Universal Robots URScript: Robot 3 12_10.script

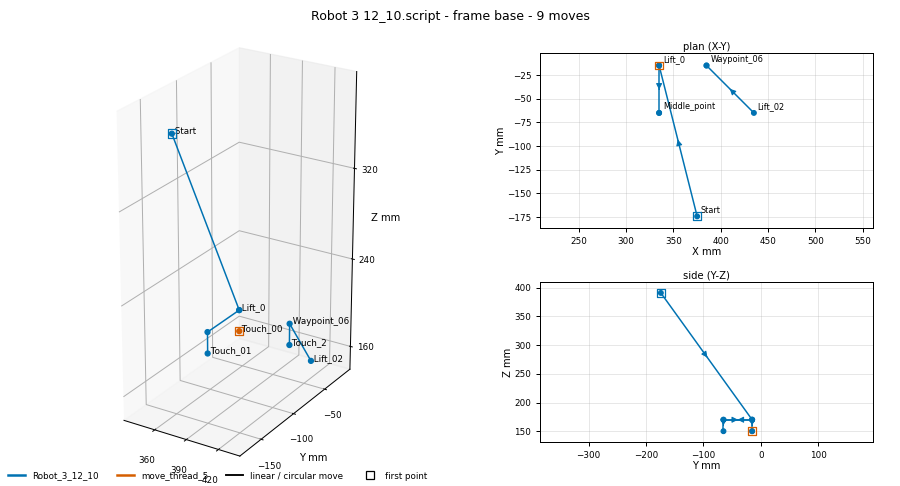
[picture p0: tool path of Robot 3 12_10.script in frame base, 9 of 16 moves have a stored position in this frame; points joined in program order, loops and branches not executed]
def Robot_3_12_10():
  set_tcp(p[0.0,0.0,0.0,0.0,0.0,0.0])
  set_safety_mode_transition_hardness(1)
  step_count_74a58e22_dc11_493a_940f_6be2cdcaf4fc = 0.0
  thread Step_Counter_Thread_ecd05ca1_44cd_422d_8c53_38ca33f79cc8():
    while (True):
      step_count_74a58e22_dc11_493a_940f_6be2cdcaf4fc = step_count_74a58e22_dc11_493a_940f_6be2cdcaf4fc + 1.0
      sync()
    end
  end
  run Step_Counter_Thread_ecd05ca1_44cd_422d_8c53_38ca33f79cc8()
  set_target_payload(0.990000, [-0.002000, -0.006000, 0.057000], [0.001514, 0.001514, 0.001514, 0.000000, 0.000000, 0.000000])
  modbus_add_signal("192.168.12.20", 255, 1001, 2, "MODBUS_1", False)
  modbus_set_signal_update_frequency("MODBUS_1", 10)
  modbus_add_signal("192.168.12.20", 255, 1003, 3, "MODBUS_2", False)
  modbus_set_signal_update_frequency("MODBUS_2", 10)
  modbus_add_signal("192.168.12.20", 255, 1005, 2, "MODBUS_3", False)
  modbus_set_signal_update_frequency("MODBUS_3", 10)
  modbus_add_signal("192.168.12.20", 255, 1008, 2, "MODBUS_4", False)
  modbus_set_signal_update_frequency("MODBUS_4", 10)
  modbus_add_signal("192.168.12.20", 255, 1007, 3, "MODBUS_5", False)
  modbus_set_signal_update_frequency("MODBUS_5", 10)
  modbus_set_runstate_dependent_choice("MODBUS_2",0)
  modbus_set_runstate_dependent_choice("MODBUS_5",0)
  set_gravity([0.0, 0.0, 9.82])
  set_tool_communication(True, 1000000, 2, 1, 1.5, 3.5)
  set_tool_output_mode(0)
  set_tool_digital_output_mode(0, 1)
  set_tool_digital_output_mode(1, 1)
  set_tool_voltage(24)
  set_standard_analog_input_domain(0, 1)
  set_standard_analog_input_domain(1, 1)
  set_tool_analog_input_domain(0, 1)
  set_tool_analog_input_domain(1, 1)
  set_analog_outputdomain(0, 0)
  set_analog_outputdomain(1, 0)
  set_input_actions_to_default()
  global Plane_1=p[0.5,0.0,0.07,-3.667604942726106E-16,3.141592653589793,-5.847522753981501E-16]
  # begin: URCap Installation Node
  #   Source: OnRobot, 5.14.0, OnRobot A/S
  #   Type: OnRobot Setup
  if (False):
  end
  ON_CONN_SHIFT_BOOL = 64
  ON_CONN_SHIFT_INT = 24
  ON_CONN_SHIFT_FLOAT = 24
  ON_CONN_REG_SUM_BOOL = 0
  ON_CONN_REG_SUM_INT = 1
  ON_CONN_REG_SUM_FLOAT = 0
  ON_TOOL_SHIFT_BOOL = 64
  ON_TOOL_SHIFT_INT = 25
  ON_TOOL_SHIFT_FLOAT = 24
  ON_TOOL_SHIFT_BOOL_ARR = [64, 64, 64]
  ON_TOOL_SHIFT_INT_ARR = [25, 25, 25]
  ON_TOOL_SHIFT_FLOAT_ARR = [24, 24, 24]
  ON_TOOL_REG_SUM_BOOL = 0
  ON_TOOL_REG_SUM_INT = 0
  ON_TOOL_REG_SUM_FLOAT = 0
  ON_REGISTERS_SPEEDL_FLOAT = 0
  ON_REG_USE_TOOL = False
  ON_DI_SINGLE = 0
  ON_DI_PRIMARY = 1
  ON_DI_SECONDARY = 2
  ON_DI_DUAL = 3
  on_robot_type = 10
  on_robot_cycle = 2.0
  on_conn_ip = "localhost"
  on_tool_ip = "localhost"
  on_device_socket_port = 51234
  on_conn_xmlrpc = rpc_factory("xmlrpc", "http://localhost:41414")
  on_tool_xmlrpc = rpc_factory("xmlrpc", "http://localhost:41414")
  on_RPC = rpc_factory("xmlrpc", "http://127.0.0.1:31416")
  ON_DEBUG_LOG = False
  on_isMetric = True
  on_toolConnector = True
  on_ioqc = False
  on_dual = False
  on_computebox = False
  on_devices = 0
  on_gripper = [False, False, False]
  on_custom_tcp_id = "none"
  on_custom_tcp_enabled = False
  on_ft = False
  #======    OnRobot Globals    ======#

  ON_MATH_PI=3.141593
  ON_ZEROPOSE=p[0.0,0.0,0.0,0.0,0.0,0.0]
  ON_ZEROFRAME=p[0.0,0.0,0.0,0.0,0.0,0.0]
  ON_ZERO3D=[0.0,0.0,0.0]
  ON_ZERO6D=[0.0,0.0,0.0,0.0,0.0,0.0]
  ON_ZERO8D=[0.0,0.0,0.0,0.0,0.0,0.0,0.0,0.0]
  ON_FALSE3D=[False,False,False]
  ON_FALSE6D=[False,False,False,False,False,False]
  ON_FALSE8D=[False,False,False,False,False,False,False,False]
  global on_return=0
  on_speedL=ON_ZERO6D
  on_speedBase=ON_ZERO6D
  on_speedVect=ON_ZERO6D
  on_speedExtra=ON_ZERO6D
  on_speedCB=ON_ZERO6D
  on_speedGecko=ON_ZERO6D
  on_RTDE_error=0
  on_RTDE_tool_error=0
  on_dataProcess_thrd=0
  ON_DEVICE_ID_MISSING=0
  ON_INIT_WATCHDOG_HZ=5
  ON_INIT_TIMEOUT=500
  on_robot_TCP_offset=ON_ZEROFRAME
  on_tcp_offset_actual=ON_ZEROFRAME
  on_cog_actual=ON_ZEROFRAME
  on_mass_actual=0.0
  on_robot_mount=[0.0,0.0]

  #======    End of OnRobot Globals    ======#
  #======    OnRobot Interface Messages    ======#

  on_devices_primary_log="OnRobot Devices"
  on_devices_secondary_log="OnRobot Secondary Device"
  on_program_halted="<br>Program halted."
  on_device_error_title="OnRobot - Device error"
  on_install_error="OnRobot Setup is not correct.<br>Check the status in the OnRobot Setup page in the Installation Tab.<br>Program halted."
  on_device_missing="No device connected.<br>Program halted."
  cb_device_missing="No OnRobot Compute Box connected.<br>Program halted."
  ft_device_missing="No OnRobot FT sensor or license detected.<br>Program halted."
  hex_device_missing="No HEX sensor connected.<br>Program halted."
  rg2ft_device_missing="No RG2-FT gripper connected.<br>Program halted."
  rg_device_missing="No RG gripper connected.<br>Program halted."
  vg_device_missing="No VG gripper connected.<br>Program halted."
  gg_device_missing="No Gecko Gripper connected.<br>Program halted."
  sg_device_missing="No Soft Gripper connected.<br>Program halted."
  tfg_device_missing="No 3FG gripper connected.<br>Program halted."
  sdr_device_missing="No OnRobot Sander connected.<br>Program halted."
  twofg_device_missing="No 2FG gripper connected.<br>Program halted."
  vgp_device_missing="No VGP gripper connected.<br>Program halted."
  mg_device_missing="No Magnetic Gripper connected.<br>Program halted."
  fgp_device_missing="No 2FGP20 Gripper connected.<br>Program halted."
  on_xmlrpc_start_ip="Connecting to OnRobot XML-RPC Server:"
  on_java_comm_error_textmsg_title="OnRobot - Communication error:"
  on_java_comm_controlsocket_open_error="Socket 'javaSocket' opening was unsuccessful."
  on_java_comm_error_title="OnRobot - Communication error"
  on_java_comm_socket_open_error="Establishing connection with the URCap was timed out.<br>Check the status in the OnRobot Setup page in the Installation Tab.<br>Program halted."
  on_rtde_feed_error_textmsg_title="OnRobot - RTDE error:"
  on_rtde_feed_error="RTDE feed error. OnRobot device count mismatch.<br>Program halted."
  on_rtde_feed_tool_error="Tool RTDE feed error. OnRobot device count mismatch.<br>Program halted."
  on_rtde_feed_open_error_textmsg="Socket 'rtdeFeed' opening was unsuccessful."
  on_rtde_feed_error_title="OnRobot - RTDE error"
  on_rtde_feed_count_error="Invalid RTDE offset setup detected. Please check RTDE Offsets at the OnRobot Setup page in the Installation Tab.<br>Program halted."
  on_rtde_feed_open_error="Establishing connection with the devices was timed out.<br>Ensure that the OnRobot devices are operational, and check the status in the OnRobot Setup page in the Installation Tab."

  #======    End of OnRobot Interface Messages    ======#
  #======    OnRobot Interface    ======#

  on_portopened_javaSocket=False
  on_rtde_feed_opened=False
  on_dataProcess_running=False
  def on_missing():
  popup(on_device_missing,title=on_device_error_title,error=True,blocking=False)
  halt
  end
  def cb_missing():
  popup(cb_device_missing,title=on_device_error_title,error=True,blocking=False)
  halt
  end
  def ft_missing():
  popup(ft_device_missing,title=on_device_error_title,error=True,blocking=False)
  halt
  end
  def hex_missing():
  popup(hex_device_missing,title=on_device_error_title,error=True,blocking=False)
  halt
  end
  def rg2ft_missing():
  popup(rg2ft_device_missing,title=on_device_error_title,error=True,blocking=False)
  halt
  end
  def rg_missing():
  popup(rg_device_missing,title=on_device_error_title,error=True,blocking=False)
  halt
  end
  def vg_missing():
  popup(vg_device_missing,title=on_device_error_title,error=True,blocking=False)
  halt
  end
  def gg_missing():
  popup(gg_device_missing,title=on_device_error_title,error=True,blocking=False)
  halt
  end
  def sg_missing():
  popup(sg_device_missing,title=on_device_error_title,error=True,blocking=False)
  halt
  end
  def tfg_missing():
  popup(tfg_device_missing,title=on_device_error_title,error=True,blocking=False)
  halt
  end
  def sdr_missing():
  popup(sdr_device_missing,title=on_device_error_title,error=True,blocking=False)
  halt
  end
  def twofg_missing():
  popup(twofg_device_missing,title=on_device_error_title,error=True,blocking=False)
  halt
  end
  def vgp_missing():
  popup(vgp_device_missing,title=on_device_error_title,error=True,blocking=False)
  halt
  end
  def mg_missing():
  popup(mg_device_missing,title=on_device_error_title,error=True,blocking=False)
  halt
  end
  def fgp_missing():
  popup(fgp_device_missing,title=on_device_error_title,error=True,blocking=False)
  halt
  end
  def on_portclose_javaSocket():
  socket_close("javaSocket")
  on_portopened_javaSocket=False
  end
  def on_portopen_javaSocket():
  on_portclose_javaSocket()
  on_portopened_javaSocket=socket_open("127.0.0.1",44005,"javaSocket")
  if not on_portopened_javaSocket:
  textmsg(on_java_comm_error_textmsg_title,on_java_comm_controlsocket_open_error)
  popup(on_java_comm_socket_open_error,title=on_java_comm_error_title,error=True,blocking=False)
  halt
  end
  end
  on_conn_rtde_feed_name="rtdeFeedConn"
  on_tool_rtde_feed_name="rtdeFeedTool"
  def on_rtde_feed_close(rtdeFeedName):
  socket_close(rtdeFeedName)
  on_rtde_feed_opened=False
  end
  def on_rtde_feed_open(deviceIP,rtdeFeedName,regStart,regSum,regSpeedl):
  on_rtde_feed_close(rtdeFeedName)
  if((regStart[0]+regSum[0])>128)or((regStart[1]+regSum[1])>48)or((regStart[2]+regSum[2])>48):
  popup(on_rtde_feed_count_error,title=on_rtde_feed_error_title,error=True,blocking=False)
  textmsg(str_cat("RegStart: ",regStart),str_cat("  -  RegSum: ",regSum))
  halt
  end
  on_rtde_feed_opened=socket_open(deviceIP,on_device_socket_port,rtdeFeedName)
  if not on_rtde_feed_opened:
  on_rtde_feed_opened=socket_open(deviceIP,on_device_socket_port,rtdeFeedName)
  end
  if not on_rtde_feed_opened:
  textmsg(on_rtde_feed_error_textmsg_title,on_rtde_feed_open_error_textmsg)
  popup(on_rtde_feed_open_error,title=on_rtde_feed_error_title,error=True,blocking=False)
  halt
  end
  socket_send_int(regStart[0],rtdeFeedName)
  socket_send_int(regSum[0],rtdeFeedName)
  socket_send_int(regStart[1],rtdeFeedName)
  socket_send_int(regSum[1],rtdeFeedName)
  socket_send_int(regStart[2],rtdeFeedName)
  socket_send_int(regSum[2],rtdeFeedName)
  socket_send_int(regSpeedl,rtdeFeedName)
  socket_send_int(on_devices,rtdeFeedName)
  end
  def on_dataRead():
  enter_critical
  on_RTDE_error=read_input_integer_register(ON_CONN_SHIFT_INT)
  if(ON_REG_USE_TOOL):
  on_RTDE_tool_error=read_input_integer_register(ON_TOOL_SHIFT_INT_ARR[0])
  end
  exit_critical
  end
  def on_set_rtde_watchdog(updateHz=ON_INIT_WATCHDOG_HZ):
  local effect="stop"
  if(updateHz<1):
  effect="ignore"
  end
  watchdog_conn_reg_str=str_cat("input_int_register_",ON_CONN_SHIFT_INT)
  rtde_set_watchdog(watchdog_conn_reg_str,updateHz,effect)
  if(ON_REG_USE_TOOL):
  watchdog_tool_reg_str=str_cat("input_int_register_",ON_TOOL_SHIFT_INT_ARR[0])
  rtde_set_watchdog(watchdog_tool_reg_str,updateHz,effect)
  end
  if ON_DEBUG_LOG:
  local update_str=str_cat(" "+effect+" watchdog set to [Hz]: ",updateHz)
  textmsg(watchdog_conn_reg_str,update_str)
  if(ON_REG_USE_TOOL):
  local update_str=str_cat(" "+effect+" watchdog set to [Hz]: ",updateHz)
  textmsg(watchdog_tool_reg_str,update_str)
  end
  end
  end
  def on_speedCB_get():
  return[on_speedCB[0],on_speedCB[1],on_speedCB[2],on_speedCB[3],on_speedCB[4],on_speedCB[5]]
  end
  def on_speedGecko_get():
  local speedExtra=ON_ZERO6D
  if on_speedl_for_gecko:
  speedExtra=[on_speedGecko[0],on_speedGecko[1],on_speedGecko[2],on_speedGecko[3],on_speedGecko[4],on_speedGecko[5]]
  end
  return speedExtra
  end
  def on_speedGecko_set(speedGecko):
  on_speedGecko=[speedGecko[0],speedGecko[1],speedGecko[2],speedGecko[3],speedGecko[4],speedGecko[5]]
  end
  thread on_dataProcess_thread():
  if ON_DEBUG_LOG:
  textmsg("Starting on_dataRead thread")
  end
  local error=False
  on_dataProcess_running=True
  sync()
  while on_dataProcess_running:
  sync()
  on_dataRead()
  error=on_error((on_RTDE_error<0),on_rtde_feed_error,on_rtde_feed_error_title,error)
  error=on_error((ON_REG_USE_TOOL and(on_RTDE_tool_error<0)),on_rtde_feed_tool_error,on_rtde_feed_error_title,error)
  on_dataProcess_running=not error
  end
  if error:
  halt
  end
  if ON_DEBUG_LOG:
  textmsg("Stopping on_dataRead thread")
  end
  end
  thread on_set_watchdog_thread():
  sleep(2)
  on_set_rtde_watchdog(updateHz=ON_INIT_WATCHDOG_HZ)
  sleep(1/ON_INIT_WATCHDOG_HZ)
  on_dataProcess_running=False
  kill on_dataProcess_thrd
  end

  #======    End of OnRobot Interface    ======#
  #======    OnRobot QC Setup Tool Connector    ======#

  def tc_setup_tool():
  if ON_DEBUG_LOG:
  textmsg("QC Setup Tool Connector start...")
  end
  set_tool_voltage(24)

  set_tool_communication(True,1000000,2,1,1.5,3.5)

  if ON_DEBUG_LOG:
  textmsg("QC Setup Tool Connector end.")
  end
  end

  #======    End of OnRobot QC Setup Tool Connector    ======#
  #======    OnRobot TCP Messages    ======#

  on_tcp_log_msg_default="OnRobot: Robot TCP Offset set to:"
  on_tcp_log_msg_primary="OnRobot: Robot TCP Offset set to Primary:"
  on_tcp_log_msg_secondary="OnRobot: Robot TCP Offset set to Secondary:"

  #======    End of OnRobot TCP Messages    ======#
  #======    OnRobot TCP    ======#

  on_tcp_offset_actual=ON_ZEROFRAME
  on_tcp_offset_primary=ON_ZEROFRAME
  on_tcp_static_primary=ON_ZEROFRAME
  on_tcp_dynamic_primary=ON_ZEROFRAME
  on_tcp_adapters=ON_ZEROFRAME
  on_tcp_qc_primary=ON_ZEROFRAME
  on_tcp_base_primary=ON_ZEROFRAME
  on_tcp_gripper_static_primary=ON_ZEROFRAME
  on_tcp_workpiece_primary=ON_ZEROFRAME
  on_tcp_gripper_dynamic_primary=ON_ZEROFRAME
  on_tcp_gripper_primary=ON_ZEROFRAME
  on_tcp_offset_secondary=ON_ZEROFRAME
  on_tcp_static_secondary=ON_ZEROFRAME
  on_tcp_dynamic_secondary=ON_ZEROFRAME
  on_tcp_qc_secondary=ON_ZEROFRAME
  on_tcp_base_secondary=ON_ZEROFRAME
  on_tcp_gripper_static_secondary=ON_ZEROFRAME
  on_tcp_workpiece_secondary=ON_ZEROFRAME
  on_tcp_gripper_dynamic_secondary=ON_ZEROFRAME
  on_tcp_gripper_secondary=ON_ZEROFRAME
  on_tcp_custom_preset_assigned=False
  on_tcp_custom_preset=ON_ZEROFRAME
  def on_tcp_init_adapters():
  if ON_DEBUG_LOG:
  textmsg("TCP Init Adapters start..")
  end
  enter_critical
  on_tcp_adapters=ON_ZEROFRAME
  local adapterCount=length(on_tcp_adapters_array)
  local i=0
  while(i<adapterCount):
  on_tcp_adapters=pose_trans(on_tcp_adapters,on_tcp_adapters_array[i])
  i=i+1
  end
  exit_critical
  if ON_DEBUG_LOG:
  textmsg("TCP Init Adapters end.")
  end
  end
  def on_tcp_update_primary():
  if ON_DEBUG_LOG:
  textmsg("TCP Update Primary start..")
  end
  on_tcp_gripper_dynamic_primary=p[0.0, 0.0, 0.0, 0.0, 0.0, 0.0]
  enter_critical
  on_tcp_dynamic_primary=pose_trans(on_tcp_static_primary,on_tcp_gripper_dynamic_primary)
  on_tcp_offset_primary=pose_trans(on_tcp_dynamic_primary,on_tcp_workpiece_primary)
  exit_critical
  if ON_DEBUG_LOG:
  textmsg("TCP Update Primary end.")
  end
  end
  def on_tcp_init_primary():
  if ON_DEBUG_LOG:
  textmsg("TCP Init Primary start..")
  end
  enter_critical
  on_tcp_base_primary=pose_trans(on_tcp_adapters,on_tcp_qc_primary)
  on_tcp_static_primary=pose_trans(on_tcp_base_primary,on_tcp_gripper_static_primary)
  exit_critical
  on_tcp_update_primary()
  if ON_DEBUG_LOG:
  textmsg("TCP Init Primary end.")
  end
  end
  def on_tcp_offset_set(TCP_offset):
  if ON_DEBUG_LOG:
  textmsg("TCP Offset set started!")
  end
  on_tcp_offset_send(TCP_offset)
  if(on_follow_tcp):
  set_tcp(TCP_offset)
  end
  on_robot_TCP_offset=TCP_offset
  if ON_DEBUG_LOG:
  textmsg("TCP Offset set to: ",on_robot_TCP_offset)
  end
  end
  def on_tcp_offset_forced_set_actual(isPrimary=True):
  if(not on_follow_tcp):

  local tcp_log_msg=on_tcp_log_msg_default

  textmsg(tcp_log_msg,on_tcp_offset_actual)
  set_tcp(on_tcp_offset_actual)
  end
  end
  def on_tcp_update(isPrimary=True):
  on_tcp_update_primary()

  on_tcp_set_actual_to(isPrimary)
  end
  def on_tcp_set_actual_to(isPrimary=True):

  on_tcp_offset_actual=on_tcp_offset_primary
  if(on_follow_tcp):
  textmsg(on_tcp_log_msg_default,on_tcp_offset_actual)
  end

  on_tcp_active_is_primary=isPrimary
  on_tcp_offset_set(on_tcp_offset_actual)
  end
  def on_tcp_update_workpiece_primary(workpiece_offset):
  if ON_DEBUG_LOG:
  textmsg("TCP Update Tool Primary start..")
  end
  on_tcp_workpiece_primary=workpiece_offset
  on_tcp_update_primary()
  if ON_DEBUG_LOG:
  textmsg("TCP Update Tool Primary end.")
  end
  end
  def on_tcp_workpiece_rpy_get(xyz=[0.0,0.0,0.0],rpy=[0.0,0.0,0.0]):
  local rotvec=rpy2rotvec(rpy)
  local workpiece_offset=p[xyz[0],xyz[1],xyz[2],rotvec[0],rotvec[1],rotvec[2]]
  return workpiece_offset
  end

  def on_tcp_update_workpiece(workpiece_offset,tool_index=0):
  if ON_DEBUG_LOG:
  textmsg("TCP Update Tool start..")
  end
  if(tool_index!=ON_DI_SECONDARY):
  on_tcp_update_workpiece_primary(workpiece_offset)
  local isPrimary=True

  end
  on_tcp_set_actual_to(isPrimary)
  if ON_DEBUG_LOG:
  textmsg("TCP Update Tool end.")
  end
  end
  def on_get_tcp_for(tool_index):
  if tool_index==ON_DI_SECONDARY:
  local actual_tcp=on_tcp_static_secondary
  else:
  local actual_tcp=on_tcp_static_primary
  end
  return actual_tcp
  end
  def on_tcp_custom_unused():
  return ON_ZEROFRAME
  end
  def on_tcp_update_custom():
  if ON_DEBUG_LOG:
  textmsg("TCP Update Custom start..")
  end
  if(on_custom_tcp_enabled):
  on_tcp_custom_unused()
  on_tcp_custom_unused()
  on_tcp_custom_unused()
  on_tcp_custom_unused()

  end
  if ON_DEBUG_LOG:
  textmsg("TCP Update Custom end.")
  end
  end

  #======    End of OnRobot TCP    ======#
  #======    OnRobot Payload Messages    ======#

  on_mass_log_msg="OnRobot: Robot Payload Mass set to:"
  on_cog_log_msg="OnRobot: Robot Payload Center of Gravity set to:"

  #======    End of OnRobot Payload Messages    ======#
  #======    OnRobot Payload    ======#

  on_cog_actual=ON_ZEROFRAME
  on_mass_actual=0.0
  on_cog_primary=ON_ZEROFRAME
  on_cog_L1L2_primary=ON_ZEROFRAME
  on_mass_primary=0.0
  on_mass_L1L2_primary=0.0
  on_cog_adapters=ON_ZEROFRAME
  on_cog_qc_primary=ON_ZEROFRAME
  on_cog_base_primary=ON_ZEROFRAME
  on_cog_gripper_primary=ON_ZEROFRAME
  on_cog_workpiece_primary=ON_ZEROFRAME
  on_mass_adapters=0.0
  on_mass_qc_primary=0.0
  on_mass_base_primary=0.0
  on_mass_gripper_primary=0.0
  on_mass_workpiece_primary=0.0
  on_cog_secondary=ON_ZEROFRAME
  on_mass_secondary=0.0
  on_cog_gripper_secondary=ON_ZEROFRAME
  on_mass_gripper_secondary=0.0
  on_cog_workpiece_secondary=ON_ZEROFRAME
  on_mass_workpiece_secondary=0.0
  ON_LB2KG001=0.45359237/100
  def on_payload_init_adapters():
  if ON_DEBUG_LOG:
  textmsg("TCP Init Adapters start..")
  end
  enter_critical
  on_cog_adapters=ON_ZEROFRAME
  on_mass_adapters=0.0
  local massLAL0Ratio=0
  local adapterAbsCOG=ON_ZEROFRAME
  local tcp_adapter_offset=ON_ZEROFRAME
  local adapterCount=length(on_tcp_adapters_array)
  local i=0
  while(i<adapterCount):
  on_mass_adapters=on_mass_adapters+on_mass_adapters_array[i]
  if(on_mass_adapters<=0):
  massLAL0Ratio=0
  else:
  massLAL0Ratio=on_mass_adapters_array[i]/on_mass_adapters
  end
  adapterAbsCOG=pose_trans(tcp_adapter_offset,on_tcp_adapters_array[i])
  adapterAbsCOG=p[adapterAbsCOG[0],adapterAbsCOG[1],adapterAbsCOG[2],0.0,0.0,0.0]
  on_cog_adapters=interpolate_pose(on_cog_adapters,adapterAbsCOG,massLAL0Ratio)
  on_cog_adapters=p[on_cog_adapters[0],on_cog_adapters[1],on_cog_adapters[2],0.0,0.0,0.0]
  tcp_adapter_offset=pose_trans(tcp_adapter_offset,on_tcp_adapters_array[i])
  i=i+1
  sync()
  end
  exit_critical
  if ON_DEBUG_LOG:
  textmsg("TCP Init Adapters end.")
  end
  end
  def on_payload_update_primary():
  if ON_DEBUG_LOG:
  textmsg("Payload Update Primary start..")
  end
  enter_critical
  on_mass_primary=on_mass_L1L2_primary+on_mass_workpiece_primary
  local massL1L2L3Ratio=on_mass_workpiece_primary/on_mass_primary
  local workpieceAbsCOG=pose_trans(on_tcp_dynamic_primary,on_cog_workpiece_primary)
  workpieceAbsCOG=p[workpieceAbsCOG[0],workpieceAbsCOG[1],workpieceAbsCOG[2],0.0,0.0,0.0]
  on_cog_primary=interpolate_pose(on_cog_L1L2_primary,workpieceAbsCOG,massL1L2L3Ratio)
  on_cog_primary=p[on_cog_primary[0],on_cog_primary[1],on_cog_primary[2],0.0,0.0,0.0]
  exit_critical
  if ON_DEBUG_LOG:
  textmsg("Payload Update Primary end.")
  end
  end
  def on_payload_init_primary():
  if ON_DEBUG_LOG:
  textmsg("Payload Init Primary start..")
  end
  enter_critical
  on_mass_base_primary=on_mass_adapters+on_mass_qc_primary
  local massL0L1Ratio=on_mass_qc_primary/on_mass_base_primary
  on_mass_L1L2_primary=on_mass_base_primary+on_mass_gripper_primary
  local massL1L2Ratio=on_mass_gripper_primary/on_mass_L1L2_primary
  local qcAbsCOG=pose_trans(on_tcp_adapters,on_cog_qc_primary)
  qcAbsCOG=p[qcAbsCOG[0],qcAbsCOG[1],qcAbsCOG[2],0.0,0.0,0.0]
  on_cog_base_primary=interpolate_pose(on_cog_adapters,qcAbsCOG,massL0L1Ratio)
  on_cog_base_primary=p[on_cog_base_primary[0],on_cog_base_primary[1],on_cog_base_primary[2],0.0,0.0,0.0]
  local gripperAbsCOG=pose_trans(on_tcp_base_primary,on_cog_gripper_primary)
  gripperAbsCOG=p[gripperAbsCOG[0],gripperAbsCOG[1],gripperAbsCOG[2],0.0,0.0,0.0]
  on_cog_L1L2_primary=interpolate_pose(on_cog_base_primary,gripperAbsCOG,massL1L2Ratio)
  on_cog_L1L2_primary=p[on_cog_L1L2_primary[0],on_cog_L1L2_primary[1],on_cog_L1L2_primary[2],0.0,0.0,0.0]
  exit_critical
  on_payload_update_primary()
  if ON_DEBUG_LOG:
  textmsg("Payload Init Primary end.")
  end
  end
  def on_payload_update():
  on_payload_update_primary()

  on_mass_actual =on_mass_primary
  on_cog_actual=on_cog_primary

  on_payload_set_actual()
  end
  def on_payload_set_actual():

  on_mass_actual =on_mass_primary
  on_cog_actual=on_cog_primary

  local CoG=[on_cog_actual[0],on_cog_actual[1],on_cog_actual[2]]
  on_payload_set(on_mass_actual,CoG)
  end
  def on_payload_update_workpiece_primary(workpiece_mass=0,workpiece_cog=[0.0,0.0,0.0]):
  if ON_DEBUG_LOG:
  textmsg("Payload Update Workpiece Primary start..")
  end
  on_cog_workpiece_primary=p[workpiece_cog[0],workpiece_cog[1],workpiece_cog[2],0.0,0.0,0.0]
  on_mass_workpiece_primary=workpiece_mass
  on_payload_update_primary()
  if ON_DEBUG_LOG:
  textmsg("Payload Update Workpiece Primary end.")
  end
  end
  def on_payload_set(mass,CoG):
  if ON_DEBUG_LOG:
  textmsg("Payload set started!")
  end
  local center_of_gravity=[CoG[0],CoG[1],CoG[2]]
  on_payload_send(center_of_gravity,mass)
  if(on_isMetric):
  local roundedMass=floor(mass*100+0.5)/100
  else:
  local roundedMass=floor(mass/ON_LB2KG001+0.5)*ON_LB2KG001
  end
  set_payload(roundedMass,center_of_gravity)
  on_mass_actual=roundedMass
  on_cog_actual=p[CoG[0],CoG[1],CoG[2],0.0,0.0,0.0]
  if ON_DEBUG_LOG:
  textmsg("Payload mass, CoG set to: ",str_cat(str_cat(mass,", "),CoG))
  end
  end

  def on_payload_update_secondary():
  end
  def on_payload_init_secondary():
  end

  def on_payload_update_workpiece(workpiece_mass,workpiece_cog=[0.0,0.0,0.0],tool_index=0):
  if ON_DEBUG_LOG:
  textmsg("Payload Update Workpiece start..")
  end
  if(tool_index!=ON_DI_SECONDARY):
  on_cog_workpiece_primary=p[workpiece_cog[0],workpiece_cog[1],workpiece_cog[2],0.0,0.0,0.0]
  on_mass_workpiece_primary=workpiece_mass
  else:
  on_cog_workpiece_secondary=p[workpiece_cog[0],workpiece_cog[1],workpiece_cog[2],0.0,0.0,0.0]
  on_mass_workpiece_secondary=workpiece_mass
  end
  on_payload_update()
  if ON_DEBUG_LOG:
  textmsg("Payload Update Workpiece end.")
  end
  end
  def on_payload_get_cog2tcp_workpiece(tool_index=0):
  if(tool_index!=ON_DI_SECONDARY):
  local cog_tool=[on_tcp_workpiece_primary[0],on_tcp_workpiece_primary[1],on_tcp_workpiece_primary[2]]
  else:
  local cog_tool=[on_tcp_workpiece_secondary[0],on_tcp_workpiece_secondary[1],on_tcp_workpiece_secondary[2]]
  end
  return cog_tool
  end

  #======    End of OnRobot Payload    ======#
  #======    OnRobot QC TCP    ======#

  onrobotmini=0

  def on_tcp_offset_send(TCP_offset):
  on_robot_TCP_offset=TCP_offset
  end
  def on_payload_send(CoG,mass):
  on_robot_payload_cog=CoG
  on_robot_payload_mass=mass
  end


  #======    End of OnRobot QC TCP    ======#
  #======    OnRobot  Speedl    ======#

  on_speedl_thread_handler=0
  on_speedl_is_enabled=False
  on_speedl_is_running=False
  on_speedl_acc=0.0
  ft_speedl_hg_caranteen_reached=False
  ft_speedl_hg_caranteen_safemode=False
  on_speedl_for_ftcontrol=False
  on_speedl_for_move=False
  on_speedl_for_handguide=False
  on_speedl_for_insertpart=False
  on_speedl_for_depthcompensation=False
  on_speedl_for_center=False
  on_speedl_for_gecko=False
  on_speedl_acc=10000.0
  on_speedl_acc_to_zero=3.0
  ON_SPEEDL_FTCONTROL=1
  ON_SPEEDL_HANDGUIDE=2
  ON_SPEEDL_TRAJECTORY=3
  ON_SPEEDL_MOVE=ON_SPEEDL_TRAJECTORY
  ON_SPEEDL_INSERTPART=4
  ON_SPEEDL_DEPTHCOMP=5
  ON_SPEEDL_CENTER=6
  ON_SPEEDL_GECKO=7
  def on_wait_ms(time_ms):
  local sync_time=ceil(norm(time_ms/2.0))
  while(sync_time>0):
  sync_time=sync_time-1
  sync()
  end
  end
  def on_error(status_flag,message,title,stop_var=False):
  if(status_flag):
  popup(message,title=title,error=True,blocking=False)
  stop_var=True
  end
  return stop_var
  end
  def on_warning(status_flag,message,title,isPopupNeeded=False,is_shown=False):
  if(status_flag):
  if(not is_shown):
  if(isPopupNeeded):
  popup(message,title=title,warning=True,blocking=False)
  else:
  textmsg(title+": ",message)
  end
  is_shown=True
  end
  else:
  is_shown=False
  end
  return is_shown
  end
  def on_speedl_add_extra(speedBase,speedExtra):
  speedSum=ON_ZERO6D
  speedBaseP=p[speedBase[0],speedBase[1],speedBase[2],speedBase[3],speedBase[4],speedBase[5]]
  speedExtraP=p[speedExtra[0],speedExtra[1],speedExtra[2],speedExtra[3],speedExtra[4],speedExtra[5]]
  speedSumP=pose_add(speedExtraP,speedBaseP)
  speedSum=[speedSumP[0],speedSumP[1],speedSumP[2],speedSumP[3],speedSumP[4],speedSumP[5]]
  return speedSum
  end

  thread on_speedl_thread():
  if ON_DEBUG_LOG:
  textmsg("Speedl thread started..")
  end
  enter_critical
  on_speedl_is_running=True
  on_speedl_is_enabled=True
  exit_critical
  on_speedL=ON_ZERO6D
  on_speedL_last=ON_ZERO6D

  while on_speedl_is_running:
  on_speedBase=on_speedCB_get()
  on_speedL=on_speedBase


  if on_speedl_is_enabled:
  if(on_speedL==ON_ZERO6D):
  on_speedL=[on_speedL_last[0]/100,on_speedL_last[1]/100,on_speedL_last[2]/100,on_speedL_last[3]/100,on_speedL_last[4]/100,on_speedL_last[5]/100]
  end
  speedl(on_speedL,a=on_speedl_acc,t=0.001)
  else:
  speedl(ON_ZERO6D,a=on_speedl_acc_to_zero,t=0.001)
  end
  on_speedL_last=on_speedL
  end

  on_speedL=ON_ZERO6D
  if ON_DEBUG_LOG:
  textmsg("Speedl thread ended.")
  end
  end
  def on_speedl_integer_get():
  local speedl_integer=binary_list_to_integer([on_speedl_for_ftcontrol,on_speedl_for_handguide,on_speedl_for_move,on_speedl_for_insertpart,on_speedl_for_depthcompensation,on_speedl_for_center,on_speedl_for_gecko])
  return speedl_integer
  end
  def on_speedl_start_for(speedl_id):
  if(speedl_id==ON_SPEEDL_FTCONTROL):
  on_speedl_for_ftcontrol=True
  elif(speedl_id==ON_SPEEDL_HANDGUIDE):
  on_speedl_for_handguide=True
  elif(speedl_id==ON_SPEEDL_TRAJECTORY):
  on_speedl_for_move=True
  elif(speedl_id==ON_SPEEDL_INSERTPART):
  on_speedl_for_insertpart=True
  elif(speedl_id==ON_SPEEDL_DEPTHCOMP):
  on_speedl_for_depthcompensation=True
  elif(speedl_id==ON_SPEEDL_CENTER):
  on_speedl_for_center=True
  elif(speedl_id==ON_SPEEDL_GECKO):
  on_speedl_for_gecko=True
  else:
  textmsg("Unknown Start speedl ID received: ",speedl_id)
  end
  local speedl_integer=on_speedl_integer_get()
  if not(speedl_integer==0):
  if not on_speedl_is_running:
  on_speedl_thread_handler=run on_speedl_thread()
  end
  end
  return on_speedl_is_running
  end
  def on_speedl_stop_for(speedl_id,brake=10,brakeRot=10):
  if(speedl_id==ON_SPEEDL_FTCONTROL):
  on_speedl_for_ftcontrol=False
  elif(speedl_id==ON_SPEEDL_HANDGUIDE):
  on_speedl_for_handguide=False
  elif(speedl_id==ON_SPEEDL_TRAJECTORY):
  on_speedl_for_move=False
  elif(speedl_id==ON_SPEEDL_INSERTPART):
  on_speedl_for_insertpart=False
  elif(speedl_id==ON_SPEEDL_DEPTHCOMP):
  on_speedl_for_depthcompensation=False
  elif(speedl_id==ON_SPEEDL_CENTER):
  on_speedl_for_center=False
  elif(speedl_id==ON_SPEEDL_GECKO):
  on_speedl_for_gecko=False
  on_speedGecko_set(ON_ZERO6D)
  else:
  textmsg("Unknown Stop speedl ID received: ",speedl_id)
  end
  local speedl_integer=on_speedl_integer_get()
  if(speedl_integer==0):
  if(on_speedl_is_running):
  kill on_speedl_thread_handler
  enter_critical
  on_speedl_is_running=False
  exit_critical

  end
  if ON_DEBUG_LOG:
  textmsg("Speedl thread stopped")
  end
  stopl(brake,brakeRot)
  end
  return on_speedl_is_running
  end
  def on_speedl_pause():
  on_speedl_is_enabled=False
  return on_speedl_integer_get()
  end
  def on_speedl_resume():
  on_speedl_is_enabled=True
  return on_speedl_integer_get()
  end

  #======    End of OnRobot  Speedl    ======#
  textmsg(on_devices_primary_log, ": Quick Changer + QC Tool Side + [0.0, 0.0, 0.0, 0.0, 0.0, 0.0]")
  on_follow_tcp = False
  on_tcp_active_is_primary = True
  on_tcp_adapters_array = []
  on_cog_adapters_array = []
  on_mass_adapters_array = []
  on_tcp_qc_primary = p[0.0, 0.0, 0.0136, 0.0, 0.0, 0.0]
  on_cog_qc_primary = p[0.0, 0.0, 0.004, 0.0, 0.0, 0.0]
  on_mass_qc_primary = 0.06
  on_tcp_gripper_static_primary = p[0.0, 0.0, 0.017, 0.0, 0.0, 0.0]
  on_cog_gripper_primary = p[0.0, 0.0, 0.002, 0.0, 0.0, 0.0]
  on_mass_gripper_primary = 0.14
  on_tcp_workpiece_primary = p[0.0, 0.0, 0.0, 0.0, 0.0, 0.0]
  on_cog_workpiece_primary = p[0.0, 0.0, 0.0, 0.0, 0.0, 0.0]
  on_mass_workpiece_primary = 0.0
  #======    OnRobot Run    ======#

  on_portopen_javaSocket()
  sync()
  textmsg(on_xmlrpc_start_ip,on_conn_ip)
  if(ON_REG_USE_TOOL):
  on_regStart_conn=[ON_CONN_SHIFT_BOOL,ON_CONN_SHIFT_INT,ON_CONN_SHIFT_FLOAT]
  on_regSum_conn=[ON_CONN_REG_SUM_BOOL,ON_CONN_REG_SUM_INT,ON_CONN_REG_SUM_FLOAT]
  on_rtde_feed_open(on_conn_ip,on_conn_rtde_feed_name,on_regStart_conn,on_regSum_conn,ON_REGISTERS_SPEEDL_FLOAT)
  sync()
  textmsg(on_xmlrpc_start_ip,on_tool_ip)
  on_regStart_tool=[ON_TOOL_SHIFT_BOOL,ON_TOOL_SHIFT_INT,ON_TOOL_SHIFT_FLOAT]
  on_regSum_tool=[ON_TOOL_REG_SUM_BOOL,ON_TOOL_REG_SUM_INT,ON_TOOL_REG_SUM_FLOAT]
  on_rtde_feed_open(on_tool_ip,on_tool_rtde_feed_name,on_regStart_tool,on_regSum_tool,0)
  sync()
  else:
  on_regStart_conn=[ON_CONN_SHIFT_BOOL,ON_CONN_SHIFT_INT,ON_CONN_SHIFT_FLOAT]
  on_regSum_conn=[ON_CONN_REG_SUM_BOOL,ON_CONN_REG_SUM_INT,ON_CONN_REG_SUM_FLOAT]
  on_rtde_feed_open(on_conn_ip,on_conn_rtde_feed_name,on_regStart_conn,on_regSum_conn,ON_REGISTERS_SPEEDL_FLOAT)
  sync()
  end
  on_set_rtde_watchdog(updateHz=0.2)
  sync()
  on_dataProcess_thrd=run on_dataProcess_thread()
  sync()
  on_tcp_init_adapters()
  on_payload_init_adapters()
  on_tcp_init_primary()
  on_payload_init_primary()

  on_tcp_update_custom()
  on_tcp_set_actual_to(on_tcp_active_is_primary)
  if(on_follow_tcp):
  on_payload_set_actual()
  end
  on_watchdog_thrd=run on_set_watchdog_thread()
  sync()

  #======    End of OnRobot Run    ======#
  #======    OnRobot QC Start    ======#

  if(on_toolConnector):
  tc_setup_tool()
  end
  sync()

  #======    End of OnRobot QC Start    ======#
  # end: URCap Installation Node
  global Start_p=p[.375126819587, -.174150000035, .391075000099, 2.221441469323, 2.221441468836, .000000000460]
  global Start_q=[-4.494804528576424E-11, -1.5707963267296607, -2.094395102184971, -4.188790205057722, -1.5707963267966765, -3.0745184176339535E-11]
  global Lift_0_p=p[.334997549857, -.015000000001, .169999998954, 2.221441423394, 2.221441422907, .000000000460]
  global Lift_0_q=[0.5013251220673194, -1.7687324791106391, -2.419742576869704, -3.665506560199573, -1.5707962659853347, 0.5013251220816101]
  global Touch_00_p=p[.335000000172, -.015000000060, .150000001030, 2.221441439521, 2.221441439033, .000000000460]
  global Touch_00_q=[0.5013210043617833, -1.8123470416322442, -2.4280614511018905, -3.613573129351826, -1.5707962862142235, 0.5013210043760393]
  def calculate_point_to_move_towards(feature, direction, position_distance):
    local posDir=[direction[0], direction[1], direction[2]]
    if (norm(posDir) < 1e-6):
      return get_target_waypoint()
    end
    local direction_vector_normalized=normalize(posDir)
    local displacement_pose=p[direction_vector_normalized[0] * position_distance,direction_vector_normalized[1] * position_distance,direction_vector_normalized[2] * position_distance,0,0,0]
    local wanted_displacement_in_base_frame=pose_sub(pose_trans(feature, displacement_pose), feature)
    return pose_add(get_target_waypoint(), wanted_displacement_in_base_frame)
  end
  global Lift_01_p=p[.334997549857, -.015000000001, .169999998954, 2.221441423394, 2.221441422907, .000000000460]
  global Lift_01_q=[0.5013251220673194, -1.7687324791106391, -2.419742576869704, -3.665506560199573, -1.5707962659853347, 0.5013251220816101]
  global Middle_point_p=p[.334997549857, -.064999999829, .169999998954, 2.221441429898, 2.221441429411, .000000000460]
  global Middle_point_q=[0.3439264152748543, -1.7772225116704927, -2.4076108172465114, -3.669148279530547, -1.5707962728249178, 0.3439264152891574]
  global Touch_01_p=p[.334997549857, -.064999999829, .150000001030, 2.221441431332, 2.221441430845, .000000000460]
  global Touch_01_q=[0.3439264138785702, -1.8201414201326305, -2.4158207570953456, -3.618019432864394, -1.5707962763054377, 0.34392641389287687]
  global Lift_02_p=p[.434997550076, -.064999999829, .169999999605, 2.221441431332, 2.221441430845, .000000000460]
  global Lift_02_q=[0.2587746770257505, -1.9071003768572208, -2.2077920836996725, -3.739089147424896, -1.5707962821117496, 0.2587746770400742]
  global Waypoint_06_p=p[.384997550136, -.014999999889, .169999999605, 2.221441443513, 2.221441443026, .000000000460]
  global Waypoint_06_q=[0.4300619165542518, -1.8374536898244713, -2.3180614858034208, -3.698466445578543, -1.570796292471603, 0.43006191656858367]
  global Touch_2_p=p[.384997550136, -.014999999889, .150000001030, 2.221441439521, 2.221441439033, .000000000460]
  global Touch_2_q=[0.43006191833755786, -1.8758956815596317, -2.3255501341486573, -3.652535803533661, -1.5707962871777452, 0.43006191835189744]
  while (True):
    $ 1 "Robot Program"
    $ 2 "MoveL"
    $ 3 "Start" "breakAfter"
    movel(Start_p, a=1.2, v=0.25)
    $ 4 "Lift_0" "breakAfter"
    movel(Lift_0_p, a=1.2, v=0.25)
    $ 5 "Touch_00" "breakAfter"
    global move_thread_flag_5=0
    thread move_thread_5():
      enter_critical
      move_thread_flag_5 = 1
      movel(Touch_00_p, a=1.2, v=0.005)
      move_thread_flag_5 = 2
      exit_critical
    end
    move_thread_flag_5 = 0
    move_thread_han_5 = run move_thread_5()
    while (True):
      local targetTcpDirection=get_target_tcp_speed()
      local stepsToRetract=tool_contact(direction=targetTcpDirection)
      if (stepsToRetract > 0):
        kill move_thread_han_5
        stopl(3.0)
        local backTrackMovement=get_actual_joint_positions_history(stepsToRetract)
        local contactPose=get_forward_kin(backTrackMovement)
        local posDir=[targetTcpDirection[0],targetTcpDirection[1],targetTcpDirection[2]]
        local retractTo=contactPose
        if (norm(posDir) > 1e-6):
          local normalizedPosDir=normalize(posDir)
          local additionalRetraction=p[normalizedPosDir[0] * -3.0E-4, normalizedPosDir[1] * -3.0E-4, normalizedPosDir[2] * -3.0E-4, 0, 0, 0]
          retractTo = pose_sub(contactPose, additionalRetraction)
        end
        movel(retractTo, a=3.0, v=0.1)
        $ 6 "Until (tool_contact_detection)"
        break
      end
      sleep(1.0E-10)
      if (move_thread_flag_5 > 1):
        join move_thread_han_5
        break
      end
      sync()
    end
    $ 7 "Direction: Base Y-"
    global move_thread_flag_7=0
    thread move_thread_7():
      enter_critical
      move_thread_flag_7 = 1
      local towardsPos=calculate_point_to_move_towards(p[0.0,0.0,0.0,0.0,0.0,0.0], [0.0,-1.0,0.0], 0.1)
      movel(towardsPos, a=1.2, v=0.25)
      move_thread_flag_7 = 2
      exit_critical
    end
    move_thread_flag_7 = 0
    move_thread_han_7 = run move_thread_7()
    while (True):
      sleep(1.0E-10)
      if (move_thread_flag_7 > 1):
        join move_thread_han_7
        $ 8 "Until (distance)"
        break
      end
      sync()
    end
    $ 9 "Direction: Base X+"
    global move_thread_flag_9=0
    thread move_thread_9():
      enter_critical
      move_thread_flag_9 = 1
      local towardsPos=calculate_point_to_move_towards(p[0.0,0.0,0.0,0.0,0.0,0.0], [1.0,0.0,0.0], 0.1)
      movel(towardsPos, a=1.2, v=0.25)
      move_thread_flag_9 = 2
      exit_critical
    end
    move_thread_flag_9 = 0
    move_thread_han_9 = run move_thread_9()
    while (True):
      sleep(1.0E-10)
      if (move_thread_flag_9 > 1):
        join move_thread_han_9
        $ 10 "Until (distance)"
        break
      end
      sync()
    end
    $ 11 "Direction: Base Y+"
    global move_thread_flag_11=0
    thread move_thread_11():
      enter_critical
      move_thread_flag_11 = 1
      local towardsPos=calculate_point_to_move_towards(p[0.0,0.0,0.0,0.0,0.0,0.0], [0.0,1.0,0.0], 0.1)
      movel(towardsPos, a=1.2, v=0.25)
      move_thread_flag_11 = 2
      exit_critical
    end
    move_thread_flag_11 = 0
    move_thread_han_11 = run move_thread_11()
    while (True):
      sleep(1.0E-10)
      if (move_thread_flag_11 > 1):
        join move_thread_han_11
        $ 12 "Until (distance)"
        break
      end
      sync()
    end
    $ 13 "Direction: Base X-"
    global move_thread_flag_13=0
    thread move_thread_13():
      enter_critical
      move_thread_flag_13 = 1
      local towardsPos=calculate_point_to_move_towards(p[0.0,0.0,0.0,0.0,0.0,0.0], [-1.0,0.0,0.0], 0.1)
      movel(towardsPos, a=1.2, v=0.25)
      move_thread_flag_13 = 2
      exit_critical
    end
    move_thread_flag_13 = 0
    move_thread_han_13 = run move_thread_13()
    while (True):
      sleep(1.0E-10)
      if (move_thread_flag_13 > 1):
        join move_thread_han_13
        $ 14 "Until (distance)"
        break
      end
      sync()
    end
    $ 15 "Lift_01" "breakAfter"
    movel(Lift_01_p, a=1.2, v=0.25)
    $ 16 "Middle_point" "breakAfter"
    movel(Middle_point_p, a=1.2, v=0.25)
    $ 17 "Touch_01" "breakAfter"
    movel(Touch_01_p, a=1.2, v=0.25)
    $ 18 "Direction: Base X+"
    global move_thread_flag_18=0
    thread move_thread_18():
      enter_critical
      move_thread_flag_18 = 1
      local towardsPos=calculate_point_to_move_towards(p[0.0,0.0,0.0,0.0,0.0,0.0], [1.0,0.0,0.0], 0.1)
      movel(towardsPos, a=1.2, v=0.25)
      move_thread_flag_18 = 2
      exit_critical
    end
    move_thread_flag_18 = 0
    move_thread_han_18 = run move_thread_18()
    while (True):
      sleep(1.0E-10)
      if (move_thread_flag_18 > 1):
        join move_thread_han_18
        $ 19 "Until (distance)"
        break
      end
      sync()
    end
    $ 20 "Lift_02" "breakAfter"
    movel(Lift_02_p, a=1.2, v=0.25)
    $ 21 "Waypoint_06" "breakAfter"
    movel(Waypoint_06_p, a=1.2, v=0.25)
    $ 22 "Touch_2" "breakAfter"
    movel(Touch_2_p, a=1.2, v=0.25)
    $ 23 "Direction: Base Y-"
    global move_thread_flag_23=0
    thread move_thread_23():
      enter_critical
      move_thread_flag_23 = 1
      local towardsPos=calculate_point_to_move_towards(p[0.0,0.0,0.0,0.0,0.0,0.0], [0.0,-1.0,0.0], 0.1)
      movel(towardsPos, a=1.2, v=0.25)
      move_thread_flag_23 = 2
      exit_critical
    end
    move_thread_flag_23 = 0
    move_thread_han_23 = run move_thread_23()
    while (True):
      sleep(1.0E-10)
      if (move_thread_flag_23 > 1):
        join move_thread_han_23
        $ 24 "Until (distance)"
        break
      end
      sync()
    end
  end
end
